FUNCTION_BLOCK FB_Logger IMPLEMENTS I_Logger
VAR_INPUT
END_VAR
VAR_OUTPUT
END_VAR
VAR
	_fileProperties	: ST_FileProperties;
END_VAR

PROPERTY FileProperties : REFERENCE TO ST_FileProperties
GET
FileProperties ref= _fileProperties;
END_GET
SET
_fileProperties := FileProperties;
END_SET
END_PROPERTY

{warning 'add method implementation '}
METHOD LogError
END_METHOD

{warning 'add method implementation '}
METHOD LogGeneric
END_METHOD

{warning 'add method implementation '}
METHOD LogInfo
END_METHOD

{warning 'add method implementation '}
METHOD LogWarning
END_METHOD

END_FUNCTION_BLOCK

(* stored: Version 1.1.0.1, ProductVersion 3.1.4024.13
   POU FB_Logger: Id {86b60fa4-cbc9-0995-00ad-63ce008210aa}, SpecialFunc None
   Property FileProperties: Id {cf4970f1-019f-0d7d-194d-eece40979b6a}
   Get Get: Id {3c4a3446-662e-0dc2-0a1b-1173128bc028}
   Set Set: Id {342e182c-81d6-0861-102e-27b46f0e464b}
   Method LogError: Id {0826df63-6e74-08c4-10be-52e84363dcaf}
   Method LogGeneric: Id {202b6ae4-7e18-0d99-16d4-423d5f5bfd54}
   Method LogInfo: Id {d4bc99de-06e2-0964-11a9-a4a87d9d7009}
   Method LogWarning: Id {8cb67f2f-1c5a-08cb-193b-66dbde75b5eb} *)
